FUNCTION_BLOCK FBALT_2_PUMPS_GRAPH
VAR_INPUT
	LS_1 : BOOL;
	LS_2 : BOOL;
	LS_3 : BOOL;
	LS_4 : BOOL;
	
END_VAR
VAR_OUTPUT
END_VAR
VAR
END_VAR

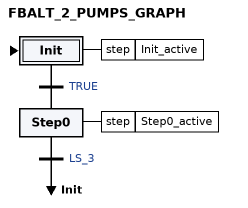
INITIAL_STEP Init:
    Init_active(N);  // step action
END_STEP
TRANSITION FROM Init TO Step0
    := TRUE;
END_TRANSITION
STEP Step0:
    Step0_active(N);  // step action
END_STEP
TRANSITION FROM Step0 TO Init
    := LS_3;
END_TRANSITION

ACTION Step0_active:
// NETWORK 1
END_ACTION

END_FUNCTION_BLOCK

(* stored: Version 1.1.0.1, ProductVersion 3.1.4024.13
   POU FBALT_2_PUMPS_GRAPH: Id {accec316-dc8f-4696-9645-26591a3dadb6}, SpecialFunc None
   Action Step0_active: Id {41422c69-8b3c-4c33-b00e-2f4b3873aac8} *)
